// TIA Portal V20 export
// export: Created 2026-04-28T10:05:09.0217582Z, ExportSetting WithDefaults, DisplayName Totally Integrated Automation Portal, DisplayVersion V20, DisplayName TIA Portal Openness, DisplayVersion V20, DisplayName TIA Portal Version Control Interface, DisplayVersion V20, DisplayName SINAMICS Startdrive Advanced, DisplayVersion V20, DisplayName SINAMICS Startdrive G130, G150, S120, S150, SINAMICS MV, G220, S200, S210, DisplayVersion V20, DisplayName SINAMICS Startdrive G110M, G120, G120C, G120D, G120P, G115D, DisplayVersion V20, DisplayName STEP 7 Professional, DisplayVersion V20, DisplayName STEP 7 Safety, DisplayVersion V20, DisplayName WinCC Basic/Comfort/Advanced, DisplayVersion V20, DisplayName WinCC Unified, DisplayVersion V20
VAR_GLOBAL   // PLC tag table "GlobVar_PLC_IO_PRG"
   x_di24VDC AT %M500.0 : Bool;   // Supply 24VDC Diagnostics 24VDC
   x_di2WayAftCy1 AT %M500.1 : Bool;   // Rohrklappenkasten nach Zyklon 1 ES4051
   x_di2WayAftCy2 AT %M500.2 : Bool;   // Rohrklappenkasten nach Zyklon 2 ES4052
   x_di2WayBin1 AT %M500.3 : Bool;   // Rohrklappenkasten unter Zyklon 1 -> Tonne ES4012
   x_di2WayBin2 AT %M500.4 : Bool;   // Rohrklappenkasten unter Zyklon 2 -> Tonne ES4022
   x_di2WayFb1 AT %M500.5 : Bool;   // Rohrklappenkasten unter Zyklon 1 -> Rückführung ES4011
   x_di2WayFb2 AT %M500.6 : Bool;   // Rohrklappenkasten unter Zyklon 2 -> Rückführung ES4021
   x_di2WayRetCy1 AT %M500.7 : Bool;   // Rohrklappenkasten Rückführung Zyklon 1 ES4041
   x_di2WayRetCy2 AT %M501.0 : Bool;   // Rohrklappenkasten Rückführung Zyklon 2 ES4042
   x_diAckBinL AT %M501.1 : Bool;   // Quittierung Fass 2 SP3011
   x_diAckBinR AT %M501.2 : Bool;   // Quittierung Fass 1 SP3012
   x_diAgitatorOnExt_1 AT %M501.3 : Bool;   // Rührwerk 1 aus extern S6009
   x_diAgitatorOffExt_1 AT %M501.4 : Bool;   // Rührwerk 1 ein extern S6010
   x_diBuFail AT %M501.5 : Bool;   // Maxon-Brenner, Störung Maxon_Stö
   x_diBuFail2 AT %M501.6 : Bool;   // Maxon-Brenner 2, Störung Maxon-2_Stö
   x_diBuOn AT %M501.7 : Bool;   // Maxon-Brenner, Ein Maxon_Ein
   x_diBuOn2 AT %M502.0 : Bool;   // Maxon-Brenner 2, eingeschaltet Maxon-2_Ein
   x_diBuOper AT %M502.1 : Bool;   // Maxon-Brenner, in Betrieb Maxon_Betr
   x_diBuOper2 AT %M502.2 : Bool;   // Maxon-Brenner 2, in Betrieb Maxon-2_Betr
   x_diCompAir AT %M502.3 : Bool;   // Druckluft Filter ES5006
   x_diEmOff AT %M502.4 : Bool;   // Not - Aus NA_PNOZ
   x_diFillBinL AT %M502.5 : Bool;   // Abfüllanlage Befüllung Fass 1 ES3011
   x_diFillBinR AT %M502.6 : Bool;   // Abfüllanlage Befüllung Fass 2 ES3012
   x_diFlyFB_1 AT %M502.7 : Bool;   // Funkenflugüberwachung Störung #1 Funkenfl_Stö_1
   x_diFlyFB_10 AT %M503.0 : Bool;   // Funkenflugüberwachung Warnung #10 Funkenfl_Warn
   x_diFlyFB_4 AT %M503.1 : Bool;   // Funkenflugüberwachung Störung #4 Funkenfl_Stö_4
   x_diFuAgitator_1 AT %M503.2 : Bool;   // Rührwerk 1 Störung FU M6052_Stö_FU
   x_diFuDeliFan AT %M503.3 : Bool;   // Schiebeventilator Störung FU M1050_Stö_FU
   x_diFuMainFa AT %M503.4 : Bool;   // Hauptventilator Störung FU M5050_Stö_FU
   x_diFuPrede AT %M503.5 : Bool;   // Staubförderventilator Störung FU M4050_Stö_FU
   x_diFuSlPump1 AT %M503.6 : Bool;   // Schlickerpumpe 1 Störung FU M6050_Stö_FU
   x_diFuSlPump2 AT %M503.7 : Bool;   // Schlickerpumpe 2 Störung FU M6051_Stö_FU
   x_diGasRate AT %M504.0 : Bool;   // Gasmenge B1004
   x_diGrGate1 AT %M504.1 : Bool;   // Granulatweiche Stellung 1 B3008/1
   x_diGrGate2 AT %M504.2 : Bool;   // Granulatweiche Stellung 2 B3008/2
   x_diMemBreak AT %M504.3 : Bool;   // Membranbruch 1 ES6001
   x_diMemBreak2 AT %M504.4 : Bool;   // Membranbruch 2 ES6002
   x_diMpAgitator_1 AT %M504.5 : Bool;   // Motorschutz Rührwerk 1 M6052_MS
   x_diMpCoBe AT %M504.6 : Bool;   // Motorschutz Förderband M3051_MS
   x_diMpDeliFan AT %M504.7 : Bool;   // Motorschutz Schiebeventilator M1050_MS
   x_diMpMainFa AT %M505.0 : Bool;   // Motorschutz Hauptventilator M5050_MS
   x_diMpPrede AT %M505.1 : Bool;   // Motorschutz Staubförderventilator M4050_MS
   x_diMpRid AT %M505.2 : Bool;   // Motorschutz Rüttelsieb M3050_MS
   x_diMpRotFe AT %M505.3 : Bool;   // Motorschutz Zellenradschleuse Zyklon M4052_MS
   x_diMpSlPump AT %M505.4 : Bool;   // Motorschutz Schlickerpumpe 1 M6050_MS
   x_diMpSlPump2 AT %M505.5 : Bool;   // Motorschutz Schlickerpumpe 2 M6051_MS
   x_diMpViCo1 AT %M505.6 : Bool;   // Motorschutz Vibrationsrinne 1 M3052_MS
   x_diMpViCo2 AT %M505.7 : Bool;   // Motorschutz Vibrationsrinne 2 M3053_MS
   x_diRetHo1 AT %M506.0 : Bool;   // Staubrückführschlauch 1 ES4031
   x_diRetHo2 AT %M506.1 : Bool;   // Staubrückführschlauch 2 ES4032
   x_diSlPuOffExt AT %M506.2 : Bool;   // Schlickerpumpe aus extern S6006
   x_diSlPuOnExt AT %M506.3 : Bool;   // Schlickerpumpe ein extern S6005
   x_diSlSuppOffExt AT %M506.4 : Bool;   // Schlickerzuführung aus extern S6008
   x_diSlSuppOnExt AT %M506.5 : Bool;   // Schlickerzuführung ein extern S6007
   x_diTwPeVaBotCl AT %M506.6 : Bool;   // Doppelpendelklappe unten geschlossen ES3016
   x_diTwPeVaBotOp AT %M506.7 : Bool;   // Doppelpendelklappe unten geöffnet ES3015
   x_diTwPeVaTopCl AT %M507.0 : Bool;   // Doppelpendelklappe oben geschlossen ES3014
   x_diTwPeVaTopOp AT %M507.1 : Bool;   // Doppelpendelklappe oben geöffnet ES3013
   x_diEmOff_60 AT %M507.2 : Bool;   // Not - Aus (Schlickerversorgung) NA_PNOZ
   x_diEmOff_10 AT %M507.3 : Bool;   // Not - Aus (Heißluftleitung) NA_PNOZ
   x_diEmOff_30 AT %M507.4 : Bool;   // Not - Aus (Austrag) NA_PNOZ
   x_diVibLimitSw_40 AT %M507.5 : Bool;   // Vibrationsgrenzschalter, Füllstand Vorentstaubung ES4060
   x_diCleanDoor AT %M507.6 : Bool;   // Reinigungstür Überwachung ES2001
   x_diVibLimitSw_50 AT %M507.7 : Bool;   // Vibrationsgrenzschalter, Füllstand Nachentstaubung ES5060
   x_diMpAgitator_2 AT %M508.0 : Bool;   // Motorschutz Rührwerk 2 M6053_MS
   x_diFuAgitator_2 AT %M508.1 : Bool;   // Rührwerk 2 Störung FU M6053_Stö_FU
   x_diMpAgitator_3 AT %M508.2 : Bool;   // Motorschutz Rührwerk 3 M6054_MS
   x_diFuAgitator_3 AT %M508.3 : Bool;   // Rührwerk 3 Störung FU M6054_Stö_FU
   x_diMpAgitator_4 AT %M508.4 : Bool;   // Motorschutz Rührwerk 4 M6055_MS
   x_diFuAgitator_4 AT %M508.5 : Bool;   // Rührwerk 4 Störung FU M6055_Stö_FU
   x_diAgitatorOnExt_2 AT %M508.6 : Bool;   // Rührwerk 2 ein extern S6011
   x_diAgitatorOffExt_2 AT %M508.7 : Bool;   // Rührwerk 2 aus extern S6012
   x_diAgitatorOnExt_3 AT %M509.0 : Bool;   // Rührwerk 3 ein extern S6013
   x_diAgitatorOffExt_3 AT %M509.1 : Bool;   // Rührwerk 3 aus extern S6014
   x_diAgitatorOnExt_4 AT %M509.2 : Bool;   // Rührwerk 4 ein extern S6015
   x_diAgitatorOffExt_4 AT %M509.3 : Bool;   // Rührwerk 4 aus extern S6016
   x_diExternSignal_1 AT %M509.4 : Bool;   // Signal 1 extern, Freigabe
   x_diSlSupp_Water AT %M509.5 : Bool;   // Endstellung Di-Wasser, Ventil Schlickerzuführung ES
   x_diSlSupp_Slip AT %M509.6 : Bool;   // Endstellung Schlicker, Ventil Schlickerzuführung ES
   x_diMpFeedWorm AT %M509.7 : Bool;   // Motorschutz Förderschnecke
   x_diManPrede AT %M510.0 : Bool;   // Staubförderventilator Handfunktion FU M43S4
   x_diMSCombAirFan AT %M510.1 : Bool;   // Motorschutz Verbrennungsluft Geblaese
   x_diHoAiTeTB45 AT %M510.2 : Bool;   // Heissluftüberwachung TB45 Ausgelöst
   x_diExAiTeTB45 AT %M510.3 : Bool;   // Abluftüberwachung TB45 Ausgelöst
   x_diPrAi AT %M510.4 : Bool;   // Dungsschalter
   x_diFillLimitSw_2 AT %M510.5 : Bool;   // Abfüllanlage Befüllung Fass 2
   x_diFillLimitSw_1 AT %M510.6 : Bool;   // Abfüllanlage Befüllung Fass 1
   x_diMainFanSpReady AT %M510.7 : Bool;   // Option Hauptventilator mit Spülung,Fertig
   x_diMpWtPuDeDust AT %M511.0 : Bool;   // Motorschutz Wasserpumpe Nassentstaubung
   x_diMpCoBe_2 AT %M511.1 : Bool;   // Motorschutz Förderband 2
   x_diTeCaFail AT %M511.2 : Bool;   // Temperaturüberwachung Schaltschrank Störung
   x_diCoBe_2_Rev_HK AT %M511.3 : Bool;   // Förderband 2 Reversieren Hardware Schalter
   x_diFillBin01 AT %M511.4 : Bool;   // Abfüllanlage Befüllung Fass 1 Schalter 52S2 Kundenspezifisch
   x_diFillBin02 AT %M511.5 : Bool;   // Abfüllanlage Befüllung Fass 2 Schalter 52S2 Kundenspezifisch
   x_diFillBin03 AT %M511.6 : Bool;   // Abfüllanlage Befüllung Fass 3 Schalter 52S2 Kundenspezifisch
   x_diFillBin04 AT %M511.7 : Bool;   // Abfüllanlage Befüllung Fass 4 Schalter 52S2 Kundenspezifisch
   x_diFillBin05 AT %M512.0 : Bool;   // Abfüllanlage Befüllung Fass 5 Schalter 52S2 Kundenspezifisch
   x_diSwMaint AT %M512.1 : Bool;   // Schlüsselschalter für Wartung Schalter 32S7.2 Kundenspezifisch
   x_diSwLaTest AT %M512.2 : Bool;   // Lampentest Schalter 33SP2 Kundenspezifisch
   x_diBuBuStart AT %M512.3 : Bool;   // Start Taster für Brenner 34SP2 Kundenspezifisch
   x_diBuBuStop AT %M512.4 : Bool;   // Stop Taster für Brenner 34S4 Kundenspezifisch
   x_diBuSlStart AT %M512.5 : Bool;   // Start Taster für Schlickerpumpe 34SP5 Kundenspezifisch
   x_diBuSlStop AT %M512.6 : Bool;   // Stop Taster für Schlickerpumpe 34S7 Kundenspezifisch
   x_diBuFaAckn AT %M512.7 : Bool;   // Störung Quittieren 34S9 Kundenspezifisch
   x_diTeCaFail_2 AT %M513.0 : Bool;   // Temperaturüberwachung Schaltschrank 2 Störung
   x_diCleanFlapOp AT %M513.1 : Bool;   // Reinigungsklappe geöffnet
   x_diCleanFlapCl AT %M513.2 : Bool;   // Reinigungsklappe geschlossen
   x_diCleanExReq AT %M513.3 : Bool;   // Reinigungseinheit Anforderderung Reinigen
   x_diCleanExFin AT %M513.4 : Bool;   // Reinigungseinheit beendet
   x_diFiFail AT %M513.5 : Bool;   // Filtersystem keine Störmeldung
   x_diFiOverTemp AT %M513.6 : Bool;   // Filtersystem Übertemperatur
   x_diFiAlarmTemp AT %M513.7 : Bool;   // Filtersystem Alarm Temperatur
   x_diCleanExFail AT %M514.0 : Bool;   // Reinigungseinheit Störung
   x_diCleanExActiv AT %M514.1 : Bool;   // Reinigungseinheit Aktiv
   x_diStartEnable AT %M514.2 : Bool;   // Freigabe Start Spruehen
   x_diSlPuEnable AT %M514.3 : Bool;   // Freigabe Schlickerpumpe
   x_diLifebit AT %M514.4 : Bool;   // Lifebit
   x_diCleanBDEActiv AT %M514.5 : Bool;   // Reinigungseinheit BDE Aktiv
   x_diCleanBDEFin AT %M514.6 : Bool;   // Reinigungseinheit BDE beendet
   x_diExtSlEmpty AT %M514.7 : Bool;   // Externe Signal Schlicker Vorrat leer
   x_diCtrlCoBe1_1 AT %M515.0 : Bool;   // Überwachung Förderband 1 B3051
   x_diCtrlCoBe1_2 AT %M515.1 : Bool;   // Überwachung Förderband 2 B3052
   x_diMainFanFlapFail AT %M515.2 : Bool;   // Klappesteuerung Hauptventilator Störung
   x_diCyFillingMax AT %M515.3 : Bool;   // Zyklon Behälter Füllstand Max B4003
   x_diBinLevelMax AT %M515.4 : Bool;   // Füllstand Pufferbehälter Max B3010
   x_diUeberCOverflow AT %M515.5 : Bool;   // Überkorn Behälter Voll
   x_diEHLimFail AT %M515.6 : Bool;   // Elektroheizung Störung Begrenzer, Störung Extern
   x_diEHTempFail AT %M515.7 : Bool;   // Elektroheizung Störung Temperartutüberwachung, Störung Extern
   x_diEHAirFail AT %M516.0 : Bool;   // Elektroheizung Störung Luftströmung, Störung Extern
   x_diEHThy1Fail AT %M516.1 : Bool;   // Elektroheizung Störung Thyristor 1, Störung Extern
   x_diEHThy2Fail AT %M516.2 : Bool;   // Elektroheizung Störung Thyristor 2, Störung Extern
   x_diHoAiTeEHTB45 AT %M516.3 : Bool;   // Heissluftüberwachung Elektroheizung TB45 Ausgelöst
   x_diPrAi_Fail AT %M516.4 : Bool;   // Dungsschalter Störmeldung
   x_diStillstand_ZSS AT %M516.5 : Bool;   // Meldung Stillstand Zerstäuberscheibe
   x_diSWErreicht_ZSS AT %M516.6 : Bool;   // Meldung Sollwert erreicht Zerstäuberscheibe
   x_diBetriebsbereit_ZSS AT %M516.7 : Bool;   // Relais Betriebsbereit Zerstäuberscheibe
   x_do2WayAftCy1a AT %M520.0 : Bool;   // Rohrklappen nach Zyklon 1a PY4051
   x_do2WayAftCy1b AT %M520.1 : Bool;   // Rohrklappen nach Zyklon 1b PY4052
   x_do2WayDuRe1 AT %M520.2 : Bool;   // Rohrklappenkasten Rückführung 1 PY4041
   x_do2WayDuRe2 AT %M520.3 : Bool;   // Rohrklappenkasten Rückführung 2 PY4042
   x_do2WayUnCy1a AT %M520.4 : Bool;   // Rohrklappen unter Zyklon 1a PY4011
   x_do2WayUnCy1b AT %M520.5 : Bool;   // Rohrklappen unter Zyklon 1b PY4012
   x_do2WayUnCy2a AT %M520.6 : Bool;   // Rohrklappen unter Zyklon 2a PY4021
   x_do2WayUnCy2b AT %M520.7 : Bool;   // Rohrklappen unter Zyklon 2b PY4022
   x_doAgitator_1 AT %M521.0 : Bool;   // Rührwerk 1 Aus/Ein M6052_A/E
   x_doBinL AT %M521.1 : Bool;   // Fass links, Leuchte SP3011
   x_doBinR AT %M521.2 : Bool;   // Fass rechts, Leuchte SP3012
   x_doBuAck AT %M521.3 : Bool;   // Maxon-Brenner, Quittieren Maxon_Quit
   x_doBudown AT %M521.4 : Bool;   // Maxon-Brenner, Brenner Kühlen Maxon_Kühlen
   x_doBuEnab AT %M521.5 : Bool;   // Maxon-Brenner, Freigabe Maxon_Freig
   x_doBuUp AT %M521.6 : Bool;   // Maxon-Brenner, Brenner Heizen Maxon_Heizen
   x_doCoBe AT %M521.7 : Bool;   // Förderband Aus/Ein M3051_A/E
   x_doDeliFan AT %M522.0 : Bool;   // Schiebeventilator Aus/Ein M1050_A/E
   x_doExAiTe AT %M522.1 : Bool;   // Abluftemperaturregelung ein Abluft_Temp_Reg
   x_doFailHo AT %M522.2 : Bool;   // Sprühtrockner Störung Hupe MFL_Hupe
   x_doFailRed AT %M522.3 : Bool;   // Sprühtrockner Störung rot MFL_Stö
   x_doFailYe AT %M522.4 : Bool;   // Sprühtrockner Vorwarnung gelb MFL_Vorw
   x_doFiSy AT %M522.5 : Bool;   // Filtersystem ein ES5009
   x_doFlySp AT %M522.6 : Bool;   // Funkenflugüberwachung Freigabe Funkenfl_Freig
   x_doFreshAir AT %M522.7 : Bool;   // Frischluftklappe PY5001
   x_doKnVa2010 AT %M523.0 : Bool;   // Klopfventil 2010 PY2010
   x_doKnVa2011 AT %M523.1 : Bool;   // Klopfventil 2011 PY2011
   x_doKnVa2012 AT %M523.2 : Bool;   // Klopfventil 2012 PY2012
   x_doKnVa2110 AT %M523.3 : Bool;   // Klopfventil 2110 PY2110
   x_doKnVa2111 AT %M523.4 : Bool;   // Klopfventil 2111 PY2111
   x_doKnVa2112 AT %M523.5 : Bool;   // Klopfventil 2112 PY2112
   x_doKnVa4061 AT %M523.6 : Bool;   // Klopfventil 4061, am Zyklon 1 PY4061
   x_doKnVa4062 AT %M523.7 : Bool;   // Klopfventil 4062, am Zyklon 2 PY4062
   x_doMainFaDelta AT %M524.0 : Bool;   // Hauptventilator (Dreieck) M5050_Dreieck
   x_doMainFan AT %M524.1 : Bool;   // Hauptventilator Aus/Ein M5050_A/E
   x_doMainFaStar AT %M524.2 : Bool;   // Hauptventilator (Stern) M5050_Stern
   x_doPrede AT %M524.3 : Bool;   // Staubförderventilator Aus/Ein M4050_A/E
   x_doReGrHuReg AT %M524.4 : Bool;   // Restfeuchteregelung ein Restf_Reg
   x_doRid AT %M524.5 : Bool;   // Rüttelsieb Aus/Ein M3050_A/E
   x_doRotFe AT %M524.6 : Bool;   // Zellenradschleuse Aus/Ein M4052_A/E
   x_doSelBinL AT %M524.7 : Bool;   // Anwahl Fass 2 PY3011
   x_doSelBinR AT %M525.0 : Bool;   // Anwahl Fass 1 PY3012
   x_doSlPump AT %M525.1 : Bool;   // Schlickerpumpe 1 Aus/Ein M6050_A/E
   x_doSlPump2 AT %M525.2 : Bool;   // Schlickerpumpe 2 Aus/Ein M6051_A/E
   x_doSlSupp AT %M525.3 : Bool;   // Schlickerzuführung ein SB6007_TL
   x_doSlSuppOnOff AT %M525.4 : Bool;   // Schlickerzuführung ein/aus PY6001
   x_doSoftReg AT %M525.5 : Bool;   // Anwahl mit Software Regler Temp
   x_doSpDrLi AT %M525.6 : Bool;   // Sprühtrockner Beleuchtung Turmbel_A/E
   x_doTwPeVaBotCl AT %M525.7 : Bool;   // Doppelpendelklappe unten schliessen PY3016
   x_doTwPeVaBotOp AT %M526.0 : Bool;   // Doppelpendelklappe unten öffnen PY3015
   x_doTwPeVaTopCl AT %M526.1 : Bool;   // Doppelpendelklappe oben schliessen PY3014
   x_doTwPeVaTopOp AT %M526.2 : Bool;   // Doppelpendelklappe oben öffnen PY3013
   x_doViCo1 AT %M526.3 : Bool;   // Vibrationsrinne 1 Aus/Ein M3052_A/E
   x_doViCo2 AT %M526.4 : Bool;   // Vibrationsrinne 2 Aus/Ein M3053_A/E
   x_doKnVa2210 AT %M526.5 : Bool;   // Klopfventil 2210 PY2210
   x_doKnVa2211 AT %M526.6 : Bool;   // Klopfventil 2211 PY2211
   x_doKnVa2212 AT %M526.7 : Bool;   // Klopfventil 2212 PY2212
   x_doKnVa5061 AT %M527.0 : Bool;   // Klopfventil 5061, am Filter 1 PY5061
   x_doKnVa5062 AT %M527.1 : Bool;   // Klopfventil 5062, am Filter 2 PY5062
   x_doAgitator_2 AT %M527.2 : Bool;   // Rührwerk 2 Aus/Ein M6053_A/E
   x_doAgitator_3 AT %M527.3 : Bool;   // Rührwerk 3 Aus/Ein M6054_A/E
   x_doAgitator_4 AT %M527.4 : Bool;   // Rührwerk 4 Aus/Ein M6055_A/E
   x_doSlSuppValve AT %M527.5 : Bool;   // Umschaltventil Schlickerzuführung PY6002
   x_doExternSignal_1 AT %M527.6 : Bool;   // Signal 1 extern, Freigabe Frisch
   x_doExternSignal_2 AT %M527.7 : Bool;   // Signal 2 extern, Überlauf
   x_doFeedWorm AT %M528.0 : Bool;   // Förderschnecke
   x_doBuSafetyCha1 AT %M528.1 : Bool;   // Sicherheit Stopp Kanal 1
   x_doBuSafetyCha2 AT %M528.2 : Bool;   // Sicherheit Stopp Kanal 2
   x_doCounterHour AT %M528.3 : Bool;   // Betriebsstundenzaehler
   x_doOmAck AT %M528.4 : Bool;   // Quittierung für PNOZ - Reset
   x_doCombAirFan AT %M528.5 : Bool;   // Verbrennungsluft Geblaese
   x_doSlCtrlHW AT %M528.6 : Bool;   // HW Regler einschalten
   x_doWtPuDeDust_On AT %M528.7 : Bool;   // Motorschutz Wasserpumpe Nassentstaubung Ein / Aus
   x_doMpCoBe_2_On AT %M529.0 : Bool;   // Motorschutz Förderband 2 Ein / Ausschalten
   x_doMpCoBe_2_Rev AT %M529.1 : Bool;   // Motorschutz Förderband 2 Reversieren
   x_doSlPumpLi AT %M529.2 : Bool;   // Schlickerpumpe externe Lampe
   x_doBetriebGr AT %M529.3 : Bool;   // Sprühtrockner Betrieb Gruen MFL_Betr
   x_doFailBl AT %M529.4 : Bool;   // Sprühtrockner Wartung Blau
   x_doLaBuBUStart AT %M529.5 : Bool;   // Lampe Start Taster für Brenner 34SP2 Kundenspezifisch
   x_doLaBuSlStart AT %M529.6 : Bool;   // Lampe Start Taster für Schlickerpumpe 34SP5 Kundenspezifisch
   x_doLaBuFaAckn AT %M529.7 : Bool;   // Lampe Störung Quittieren 34S9 Kundenspezifisch
   x_doCleanFlapOp AT %M530.0 : Bool;   // Reinigungsklappe öffnen
   x_doCleanFlapCl AT %M530.1 : Bool;   // Reinigungsklappe schliessen
   x_doCleanExReady AT %M530.2 : Bool;   // Sprühtrockner bereit
   x_doMainFanOpen AT %M530.3 : Bool;   // Abluftklappe öffnen Hauptventilator
   x_doMainFanClose AT %M530.4 : Bool;   // Abluftklappe Schliessen Hauptventilator
   x_doCleanExAckn AT %M530.5 : Bool;   // Externe Reinigung Quittierung
   x_doCleanExRes AT %M530.6 : Bool;   // Externe Reinigung Reserve
   x_doKnVa2013 AT %M530.7 : Bool;   // Klopfventil 2013 PY2013
   x_doFiVa5011 AT %M531.0 : Bool;   // Filterreinigung Ventil 5011 PY5011
   x_doFiVa5012 AT %M531.1 : Bool;   // Filterreinigung Ventil 5012 PY5012
   x_doFiVa5013 AT %M531.2 : Bool;   // Filterreinigung Ventil 5013 PY5013
   x_doFiVa5014 AT %M531.3 : Bool;   // Filterreinigung Ventil 5014 PY5014
   x_doFiVa5015 AT %M531.4 : Bool;   // Filterreinigung Ventil 5015 PY5015
   x_doFiVa5016 AT %M531.5 : Bool;   // Filterreinigung Ventil 5016 PY5016
   x_doMaOpActiv AT %M531.6 : Bool;   // Betriebsart Einrichten aktiv
   x_doAutoOpRunning AT %M531.7 : Bool;   // Betriebsart Automatik in Betrieb
   x_doCleanReq AT %M532.0 : Bool;   // Reinigung Anforderung
   x_doCleanReqFlapOp AT %M532.1 : Bool;   // Reinigungsklappe öffnen Anforderung
   x_doMaFailure AT %M532.2 : Bool;   // Anlage in Störung
   x_doLifebit AT %M532.3 : Bool;   // Lifebit
   x_doSlPuRunning AT %M532.4 : Bool;   // Externe Signal schlickerpumpe gestartet
   x_doPolyCoOn AT %M532.5 : Bool;   // Polyförderer Ein/Aus PY3017
   x_doPolyCoOn_2 AT %M532.6 : Bool;   // 2. Polyförderer Ein/Aus PY3018
   x_doProAirAvailable AT %M532.7 : Bool;   // Prozessluft Vorhanden
   x_doOnOff_ZSS AT %M533.0 : Bool;   // Start-Stopp Zerstäuberscheibe
   x_doCounterHour20 AT %M533.1 : Bool;   // Betriebsstundenzaehler D20
   x_doBuEnab2 AT %M533.2 : Bool;   // Maxon-Brenner, Freigabe Maxon_Freig D20
   x_doBuAck2 AT %M533.3 : Bool;   // Maxon-Brenner, Quittieren Maxon_Quit D20
   x_do_PwViVent AT %M533.4 : Bool;   // Magnetventil für Vibrationsbelüfter S02
   x_do_PwViMot AT %M533.5 : Bool;   // Elektrovibrator M1
   x_do_RotFi AT %M533.6 : Bool;   // Zellenradschleuse Aus/Ein Filter M5052_A/E
   x_do_VaSwFlap AT %M533.7 : Bool;   // Ventil Umschaltung Klappe öffnen
   di_aiAgitator_1 AT %MW535 : Word;   // Rührwerk 1 Istwert M6052_Ist
   di_aiCoAi AT %MW537 : Word;   // Luftmenge Düse HB6010
   di_aiDeliFan AT %MW539 : Word;   // Schiebeventilator Istwert M1050_Ist
   di_aiDiDuFiBa AT %MW541 : Word;   // Differenzdruck Filter, Staubförderventilator HB4001
   di_aiDiFiBurn AT %MW543 : Word;   // Differenzdruck Brenner HB1006
   di_aiDiPrFi AT %MW545 : Word;   // Differenzdruck Filter HB5005
   di_aiDuFiMo AT %MW547 : Word;   // Staubfilter Überwachung HB5007
   di_aiExAiTe AT %MW549 : Word;   // Ablufttemperatur Istwert D5003
   di_aiFlRa AT %MW551 : Word;   // Massedurchfluss (Schlickermenge) HB6004
   di_aiFlRaAirBurn AT %MW553 : Word;   // Zufuhr Volumenstrom Brenner HB1007/2
   di_aiFlRaAirFlue AT %MW557 : Word;   // Luftvolumenstrom Kamin HB5008/1
   di_aiFlRaAirPrede AT %MW559 : Word;   // Luftvolumenstrom Staubrückführung HB4002/1
   di_aiGrTe AT %MW561 : Word;   // Granulattemperatur B3001
   di_aiHoAiTe AT %MW563 : Word;   // Heisslufttemperatur Istwert B1001_Ist
   di_aiMainFan AT %MW565 : Word;   // Hauptventilator Istwert M5050_Ist
   di_aiMoCu AT %MW567 : Word;   // Hauptventilator Istwert Stomaufnahme M5050_Ist_Strom
   di_aiPrAi AT %MW569 : Word;   // Druck Zerstäubungsluft HB6011
   di_aiPrCy AT %MW571 : Word;   // Unterdruck im Zyklon (Abluft) HB5003
   di_aiPrede AT %MW573 : Word;   // Staubförderventilator Istwert M4050_Ist
   di_aiPrSl AT %MW575 : Word;   // Schlickerdruck HB6003
   di_aiPrTo AT %MW577 : Word;   // Unterdruck im Turm HB2003
   di_aiReGrHu AT %MW579 : Word;   // Granulatrestfeuchte HB3002
   di_aiScaleL AT %MW581 : Word;   // Waage 2 Istwert HB3006
   di_aiScaleR AT %MW583 : Word;   // Waage 1 Istwert HB3005
   di_aiSlPump1 AT %MW585 : Word;   // Schlickerpumpe 1 Istwert M6050_Ist
   di_aiSlPump2 AT %MW587 : Word;   // Schlickerpumpe 2 Istwert M6051_Ist
   di_aiSlRes AT %MW589 : Word;   // Schlickervorratsbehälter HB6008
   di_aiSpDrTe1 AT %MW591 : Word;   // Temperatur Level 1 B2010
   di_aiSpDrTe2 AT %MW593 : Word;   // Temperatur Level 2 D2011
   di_aiSpDrTe3 AT %MW597 : Word;   // Temperatur Level 3 D2012
   di_aiSpDrTe4 AT %MW599 : Word;   // Temperatur Level 4 D2013
   di_aiTempBurn AT %MW601 : Word;   // Zufuhr Temperatur Brenner HB1007/1
   di_aiTempFlue AT %MW603 : Word;   // Zuführtemperatur Kamin HB5008/2
   di_aiTempPrede AT %MW605 : Word;   // Zuführtemperatur Staubrückführung HB4002/2
   di_aiDiPrSucFi AT %MW607 : Word;   // Differenzdruck Nachfilter HB5006
   di_aiHeatExIn AT %MW609 : Word;   // Temp. Wärmetauscher Eintritt D5010
   di_aiHeatExOut AT %MW611 : Word;   // Temp. Wärmetauscher Austritt D5011
   di_aiAgitator_2 AT %MW613 : Word;   // Rührwerk Istwert 2 M6053_Ist
   di_aiAgitator_3 AT %MW615 : Word;   // Rührwerk Istwert 3 M6054_Ist
   di_aiAgitator_4 AT %MW617 : Word;   // Rührwerk Istwert 4 M6055_Ist
   di_aiScaleAgitator_1 AT %MW619 : Word;   // Waage Rührwerksbehälter 1 HB6021
   di_aiScaleAgitator_2 AT %MW621 : Word;   // Waage Rührwerksbehälter 2 HB6022
   di_aiScaleAgitator_3 AT %MW623 : Word;   // Waage Rührwerksbehälter 3 HB6023
   di_aiScaleAgitator_4 AT %MW625 : Word;   // Waage Rührwerksbehälter 4 HB6024
   di_aiOelTemp AT %MW627 : Word;   // Öltemperatur Schlickerpumpe D6030
   di_aiTempCoolWater AT %MW629 : Word;   // Temperatur Kühlwasser B
   di_aiFlowCoolWater AT %MW631 : Word;   // Durchflusswächter Kühlwasser B
   di_aiGasRate AT %MW633 : Word;   // Gaszähler D400
   di_aiPrSl2 AT %MW635 : Word;   // Schlickerdruck 2 HB6005
   di_aiSlPuControl AT %MW637 : Word;   // Schlickerdruck Druckregelung
   di_aiViscosity1 AT %MW639 : Word;   // Viskositätsmessung 1
   di_aiViscosity2 AT %MW641 : Word;   // Viskositätsmessung 2
   di_aiTempSl AT %MW643 : Word;   // Schlickertemperatur
   di_aiViscoTemp AT %MW645 : Word;   // Temperatur bei der Viskositätsmessung 1
   di_aiLeMonitor AT %MW647 : Word;   // Füllstandsüberwachung am Pulverbehälter
   di_aiMainFanPosFlap AT %MW649 : Word;   // Stellglied der Klappe auf/zu
   di_aiFlProAir AT %MW651 : Word;   // Prozessluft Menge
   di_aiPrCompAir AT %MW653 : Word;   // Druckluft Filteranlage
   di_aiPrFiBefore AT %MW655 : Word;   // Unterdruckschalter Ansaugfilter Vor
   di_aiPrFiAfter AT %MW657 : Word;   // Unterdruckschalter Nach Filter
   di_aiFlRaCy AT %MW659 : Word;   // Strömungsüberwachung Staubrückführung HB4003
   di_aoAgitator_1 AT %MW661 : Word;   // Rührwerk 1 Sollwert M6052_Soll
   di_aoDeliFan AT %MW663 : Word;   // Schiebeventilator Sollwert M1050_Soll
   di_aoExAiTe AT %MW665 : Word;   // Ablufttemperatur Sollwert Abluft-Temp_Soll
   di_aoHoAir AT %MW667 : Word;   // Heißlufttemperatur Sollwert HL-Temp_Soll
   di_aoMainFan AT %MW669 : Word;   // Hauptventilator Sollwert M5050_Soll
   di_aoPrede AT %MW671 : Word;   // Staubförderventilator Sollwert M4050_Soll
   di_aoReGrHu AT %MW673 : Word;   // Restfeuchteregelung Sollwert Restfeuchte_Soll
   di_aoSlPump AT %MW675 : Word;   // Schlickerpumpe 1 Sollwert M6050_Soll
   di_aoSlPump2 AT %MW677 : Word;   // Schlickerpumpe 2 Sollwert M6051_Soll
   di_aoAgitator_2 AT %MW679 : Word;   // Rührwerk 2 Sollwert M6053_Soll
   di_aoAgitator_3 AT %MW681 : Word;   // Rührwerk 3 Sollwert M6054_Soll
   di_aoAgitator_4 AT %MW683 : Word;   // Rührwerk 4 Sollwert M6055_Soll
   di_aoLevelAgitator_1 AT %MW685 : Word;   // Istwert Füllstand Rührwerksbehälter 1
   di_aoLevelAgitator_2 AT %MW687 : Word;   // Istwert Füllstand Rührwerksbehälter 2
   di_aoLevelAgitator_3 AT %MW689 : Word;   // Istwert Füllstand Rührwerksbehälter 3
   di_aoLevelAgitator_4 AT %MW691 : Word;   // Istwert Füllstand Rührwerksbehälter 4
   di_aoSlPuControl AT %MW693 : Word;   // Schlickerdruck Druckregelung FU
   di_aoMainFanSetFlap AT %MW695 : Word;   // Sollwert Stellung der Klappe
   x_diSicherheitSchalter_ZSS AT %M517.0 : Bool;   // Sicherheitsschalter Gerät im Position
   di_aoSollwert_ZSS AT %MW697 : Word;   // Sollwert Zerstäuberscheibe
   di_aiIstwert_ZSS AT %MW699 : Word;   // Frequez-Istwert Zerstäuberscheibe
   di_aiTeEH_TB45 AT %MW701 : Word;   // Temperature from the electric heater via the TB45 shutdown precondition for the main fan
   di_aiTeEH_PwAkt AT %MW703 : Word;   // Power measurement from the electric heater Signal from the heater
   x_diRidOverflow AT %M517.1 : Bool;
   di_aiExAiTeD20 AT %MW705 : Word;   // Ablufttemperatur Istwert D5003 D20
   di_aiHoAiTeD20 AT %MW707 : Word;   // Heisslufttemperatur Istwert B1001_Ist D20
   di_aiPrCyD20 AT %MW709 : Word;   // Unterdruck im Zyklon (Abluft) HB5003 D20
   di_aiPrToD20 AT %MW711 : Word;   // Unterdruck im Turm HB2003 D20
   di_aiGasRateD20 AT %MW713 : Word;   // Gaszähler D20
   di_aiPrSlD20 AT %MW715 : Word;   // Schlickerdruck HB6003 D20
   di_aiFlRaD20 AT %MW717 : Word;   // Massedurchfluss (Schlickermenge) HB6004 D20
   x_diPwLeSw AT %M517.2 : Bool;   // Fuellstandsensor am Pulverzufuehrung S01
   di_aoHoAirD20 AT %MW719 : Word;   // Heißlufttemperatur Sollwert HL-Temp_Soll D20
   x_diMpRotFilter AT %M517.3 : Bool;   // Motorschutz Zellenradschleuse FilterM5052_MS
   x_diMemBreak3 AT %M517.4 : Bool;   // Membranbruch 3 ES6003
   x_diFiMonEmpty AT %M517.5 : Bool;   // Filteranlage Überwachung Niveau Sensor Leer B5060
   x_diFiMonFull AT %M517.6 : Bool;   // Filteranlage Überwachung Niveau Sensor Voll B5061
   x_diFiMonRotaryFi AT %M517.7 : Bool;   // Filteranlage Überwachung Zellenrad Filter B5062
   x_diFiMonRotaryCy AT %M518.0 : Bool;   // Filteranlage Überwachung Zellenrad Zyklon B4053
   x_diEnable AT %M518.1 : Bool;   // Schlüsselschalter Eingaben erlaubt
   x_doVaSwFlapOpen AT %M533.7 : Bool;   // Ventil Umschaltung Klappe öffnen
   x_diVaSwFlapOpen AT %M518.2 : Bool;   // Ventil Umschaltung Klappe öffnen
   x_diVaSwFlapClose AT %M518.3 : Bool;   // Ventil Umschaltung Klappe schliessen
   x_doVaSwFlapClose AT %M534.0 : Bool;   // Ventil Umschaltung Klappe Schliessen
END_VAR
